{attribute 'GeneratedUsingTerminal: EP9128-0020-0016'}
{attribute addProperty BoxType "EP9128-0020-0016"}
{attribute addProperty Id "A_0004_EP9128_0021_0016A_0004_EP9128_0021_0016_AE37069D533A_0001_EP9128_0020_0016_2_EP9128_1020EP9128_1FC0878B2A_0001_EP9128_0020_0016_3_EP9128_2020EP9128_1FC0878B2"}
{attribute addProperty CRC "3287702187"}
{attribute addProperty Size "537"}
TYPE A_0001_EP9128_0020_0016_C3F65AAB EXTENDS EP9128_1FC0878B :
STRUCT
	{attribute addProperty Name "A_0004_EP9128_0021_0016"}
	{attribute addProperty PreviousPort "A_0001(EP9128-0020-0016) : D"}
	A_0004_EP9128_0021_0016 : A_0004_EP9128_0021_0016_AE37069D;
	{attribute addProperty Name "A_0001_EP9128_0020_0016_2_EP9128_1020"}
	{attribute addProperty PreviousPort "A_0001(EP9128-0020-0016) : C"}
	A_0001_EP9128_0020_0016_2_EP9128_1020 : EP9128_1FC0878B;
	{attribute addProperty Name "A_0001_EP9128_0020_0016_3_EP9128_2020"}
	{attribute addProperty PreviousPort "A_0001(EP9128-0020-0016)_2 (EP9128-1020) : C"}
	A_0001_EP9128_0020_0016_3_EP9128_2020 : EP9128_1FC0878B;
END_STRUCT
END_TYPE

(* stored: Version 1.2.0.0, ProductVersion 3.1.4024.9
   DUT A_0001_EP9128_0020_0016_C3F65AAB: Id {bebf1086-3b18-45c7-ab76-a0fb44de02ea} *)
